TYPE OffsetSicurezzaIngombro :
STRUCT
	X: Offset_Sicurezza;
	Y: Offset_Sicurezza;
	Z: Offset_Sicurezza;
	J: Offset_Sicurezza;
END_STRUCT
END_TYPE

(* stored: Version 1.1.0.1, ProductVersion 3.1.4024.11
   DUT OffsetSicurezzaIngombro: Id {3f593820-d88e-4dfa-a46c-23d8c171a263} *)
